FUNCTION_BLOCK FB_MPS_STATES
VAR_INPUT
	GANTRY    : HOMS_GANTRY;         //The horizontal gantry we are controlling
	OUT_LS    : BOOL;                //The limit switch we will travel to the out position on
	IN_RANGE  : ARRAY[0..1] OF DINT; //The range considered inserted   
	OUT_RANGE  : ARRAY[0..1] OF DINT; //The range considered inserted   
END_VAR
VAR_OUTPUT
	IN  :  BOOL; 
	OUT :  BOOL;
END_VAR
VAR
	IN_POS  : BOOL;
	OUT_POS : BOOL;
END_VAR

(* *)
//Check inserted condition
///////////////////////////////////
IN_POS := IN_RANGE[0] <= GANTRY.PAxis.diEncCnt
		  AND GANTRY.PAxis.diEncCnt < IN_RANGE[1];

//Check removed condition
////////////////////////////////////
OUT_POS := OUT_RANGE[0] <= GANTRY.PAxis.diEncCnt	
		  AND GANTRY.PAxis.diEncCnt < OUT_RANGE[1];

//Report state, not allowing both to be active
///////////////////////////////////////////////
IN := IN_POS  AND NOT OUT_POS;
OUT:= OUT_POS AND NOT IN_POS;

END_FUNCTION_BLOCK

(* stored: Version 1.1.0.1, ProductVersion 3.1.4024.6
   POU FB_MPS_STATES: Id {d3857905-9b10-40fa-a316-c3084fbb860f}, SpecialFunc None *)
